FUNCTION_BLOCK differential (* Restrained differential protection device *)
  (* Standard: IEC 61499; ApplicationDomain: AUT EMSOFT *)
  (* Version 1.0, 2021-03-23, Badger, AUT EMSOFT *)
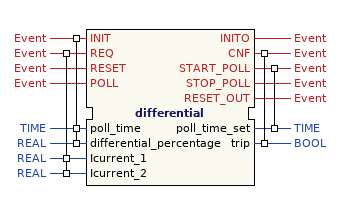
  EVENT_INPUT
    INIT WITH differential_percentage, poll_time; (* Initialization Request *)
    REQ WITH Icurrent_1, Icurrent_2; (* Normal Execution Request *)
    RESET;
    POLL;
  END_EVENT
  EVENT_OUTPUT
    INITO; (* Initialization Confirm *)
    CNF WITH trip; (* Execution Confirmation *)
    START_POLL WITH poll_time_set; (* Start the poll cycle for the differential current sampling *)
    STOP_POLL; (* Stop *)
    RESET_OUT;
  END_EVENT
  VAR_INPUT
    poll_time : TIME; (* Polling time for sampling the current differential in ms. *)
    differential_percentage : REAL; (* Input event qualifier *)
    Icurrent_1 : REAL; (* Measured current one *)
    Icurrent_2 : REAL; (* Measured current 2 *)
  END_VAR
  VAR_OUTPUT
    poll_time_set : TIME; (* Output event qualifier *)
    trip : BOOL;
  END_VAR
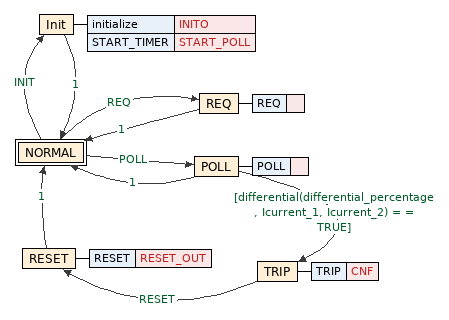
  EC_STATES
    NORMAL; (* Initial State *)
    Init : initialize -> INITO, START_TIMER -> START_POLL; (* Initialization *)
    REQ : REQ;
    POLL : POLL;
    TRIP : TRIP -> CNF;
    RESET : RESET -> RESET_OUT;
  END_STATES
  EC_TRANSITIONS
    NORMAL TO Init := INIT; (* Initialise *)
    Init TO NORMAL := 1;
    NORMAL TO REQ := REQ;
    REQ TO NORMAL := 1;
    NORMAL TO POLL := POLL;
    POLL TO TRIP := [differential(differential_percentage , Icurrent_1, Icurrent_2) = = TRUE];
    TRIP TO RESET := RESET;
    RESET TO NORMAL := 1;
    POLL TO NORMAL := 1;
  END_TRANSITIONS
  ALGORITHM initialize IN AnyText: (* Initialization algorithm *)
	cout << "alg_initialise\n";
  END_ALGORITHM
  ALGORITHM START_TIMER IN AnyText: (* new algorithm *)
	cout << "algSTART_TIMER\n";
  END_ALGORITHM
  ALGORITHM REQ IN AnyText: (* new algorithm *)
	cout << "algREQ\n";
  END_ALGORITHM
  ALGORITHM POLL IN AnyText: (* new algorithm *)
	cout << "algPOLL\n";
  END_ALGORITHM
  ALGORITHM RESET IN AnyText: (* new algorithm *)

  END_ALGORITHM
  ALGORITHM TRIP IN AnyText: (* new algorithm *)

  END_ALGORITHM
  ALGORITHM differential IN AnyText: (* calculates the differential between the currents *)
	cout << "algdifferential";
  END_ALGORITHM
END_FUNCTION_BLOCK
